FUNCTION_BLOCK AUI_LE (* less or equal *)
  (* Standard: 61131-3; Classification: standard comparison function; Description: Copyright (c) 2013 TU Wien ACIN This program and the accompanying materials are made available under the terms of the Eclipse Public License 2.0 which is available at https://www.eclipse.org/legal/epl-2.0/ SPDX-License-Identifier: EPL-2.0 *)
  (* Version 3.0, 2025-04-14, Patrick Aigner, changed package *)
  (* Version 1.0, 2013-03-13, Monika Wenger, TU Wien ACIN *)
  PACKAGE adapter::iec61131::comparison;
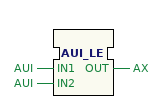
  SOCKETS
    IN1 : adapter::types::unidirectional::AUI; (* Input value 1 *)
    IN2 : adapter::types::unidirectional::AUI; (* Input value 2 *)
  END_SOCKETS
  PLUGS
    OUT : adapter::types::unidirectional::AX; (* value 1 <= value2 = true *)
  END_PLUGS
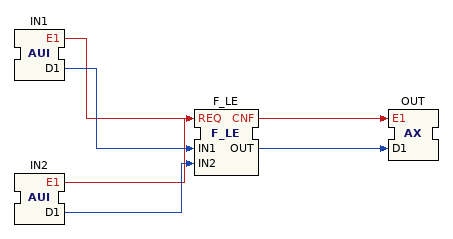
  FBS
    F_LE : iec61131::comparison::F_LE;
  END_FBS
  EVENT_CONNECTIONS
    F_LE.CNF TO OUT.E1;
    IN1.E1 TO F_LE.REQ;
    IN2.E1 TO F_LE.REQ;
  END_CONNECTIONS
  DATA_CONNECTIONS
    F_LE.OUT TO OUT.D1;
    IN1.D1 TO F_LE.IN1;
    IN2.D1 TO F_LE.IN2;
  END_CONNECTIONS
END_FUNCTION_BLOCK
